Fanuc KAREL source: kd00053.KL

-- PROVISIONAL review KL for V1013-1; original PC SHA256 e8484663d6c8198d14edd343156e697419479f5f488ecfd5bc483aa82442f582
-- Incomplete behavior may be omitted. Consult companion uncertainty JSON. Do not deploy.
PROGRAM KD00053
%NOLOCKGROUP
VAR
  I : INTEGER
  J : INTEGER
  B : BOOLEAN
  R : REAL
  S : STRING[80]
BEGIN
  -- UNRESOLVED_PC offsets 5-19; opcodes 21,9D,52,23
  -- UNRESOLVED_PC offsets 24-28; opcodes 7F
END KD00053
